// PackagingMachine object represents the packaging machine as a whole.

// right now though the packaging machine only consists of staubli robot,
// but in future projects of extending the system it is now "easy" to do so.

FUNCTION_BLOCK PackagingMachine EXTENDS UnitBaseClass
VAR_INPUT
	// initialization inputs
	inputMode		:	E_PMLProtectedUnitMode;
	inputCommand	:	E_PMLCommand;
	
	// buttons for state changes. only 6 can be used though (6 buttons in kapula)
	resetButton		AT %I*:	BIT;
	startButton		AT %I*:	BIT;
	stopButton		AT %I*:	BIT;
	holdButton		AT %I*:	BIT;
	unHoldButton	AT %I*:	BIT;
	suspendButton	AT %I*:	BIT;
	unSuspendButton	AT %I*:	BIT;
	abortButton		AT %I*:	BIT;
	clearButton		AT %I*:	BIT;
	
	// mode change buttons
	productionModeButton	AT %I*:	BIT;
	maintenanceModeButton	AT %I*:	BIT;
	manualModeButton		AT %I*:	BIT;
	
END_VAR
VAR_OUTPUT
	
END_VAR
VAR
	// container for subunits. atm only 1 subunit.
	subUnits	:	POINTER TO ARRAY[1..CONST_GV.nSubUnits] OF UnitBaseClass	:=	0;
	
	//counter for initialization
	i	:	INT;
END_VAR

IF NOT initialized THEN
	SUPER^(modeCommand:=inputMode, command:=inputCommand);
	
	IF subUnits = 0 THEN
		// subUnitsError, call setSubUnits() before PackagingMachine()
		RETURN;
	END_IF
	
	FOR i:=1 TO CONST_GV.nSubUnits BY 1 DO
		// if any of the sub units is uninitialized then the whole machine is too
		IF NOT subUnits^[i].initialized THEN
			THIS^.initialized := FALSE;
		END_IF
	END_FOR
END_IF

METHOD getSignal : INT
VAR_INPUT
END_VAR

// arranged in a way that most important ones are checked first.

// probably needs more conditions than just button signal pressed. 
// for example the statements should be ignored if machine in transition state etc.

IF abortButton THEN
	getSignal := abortSignal;
	RETURN;
	
ELSIF stopButton THEN
	getSignal := stopSignal;
	RETURN;
	
ELSIF startButton THEN
	getSignal := startSignal;
	RETURN;
	
ELSIF resetButton THEN
	getSignal := resetSignal;
	RETURN;
	
ELSIF clearButton THEN
	getSignal := clearSignal;
	RETURN;
	
ELSIF holdButton THEN
	getSignal := holdSignal;
	RETURN;
	
ELSIF unHoldButton THEN
	getSignal := unHoldSignal;
	RETURN;
	
ELSIF suspendButton THEN
	getSignal := suspendSignal;
	RETURN;
	
ELSIF unSuspendButton THEN
	getSignal := unSuspendSignal;
	RETURN;

ELSIF productionModeButton THEN
	getSignal := productionModeSignal;
	RETURN;
	
ELSIF maintenanceModeButton THEN
	getSignal := maintenanceModeSignal;
	RETURN;
	
ELSIF manualModeButton THEN
	getSignal := manualModeSignal;
	RETURN;
	
ELSE
	getSignal := -1;
	
END_IF
END_METHOD

METHOD setMode : BOOL
VAR_INPUT
	modeCommand	:	DINT;
END_VAR
VAR
	prevMode	:	E_PMLProtectedUnitMode;
END_VAR
// if any of the subUnits cannot change mode to given mode return false
FOR i:=1 TO CONST_GV.nSubUnits BY 1 DO
	IF NOT subUnits^[i].setMode(modeCommand:=modeCommand) THEN
		setMode := FALSE;
		RETURN;
	END_IF
END_FOR
SUPER^.setMode(modeCommand:=modeCommand);
setMode := TRUE;
END_METHOD


// setState method. Attempts to change the state of unit according to 
// the given input command which is a result of received user signal (startButton, stopButton ... ).

(* possible commands :	
	ePMLCommand_Undefined   := 0,
	ePMLCommand_Reset       := 1,
	ePMLCommand_Start       := 2,
	ePMLCommand_Stop        := 3,
	ePMLCommand_Hold        := 4,
	ePMLCommand_Unhold      := 5,
	ePMLCommand_Suspend     := 6,
	ePMLCommand_Unsuspend   := 7,
	ePMLCommand_Abort       := 8,
	ePMLCommand_Clear       := 9
*)

METHOD setState : BOOL
VAR_INPUT
	command	:	E_PMLCommand;
END_VAR
VAR
	prevState	:	E_PMLState;
	i			:	INT;
END_VAR
// if any of the subUnits cannot change state to given state return false
FOR i:=1 TO CONST_GV.nSubUnits BY 1 DO
	IF NOT subUnits^[i].setState(command:=command) THEN
		setState := FALSE;
		RETURN;
	END_IF
END_FOR
SUPER^.setState(command:=command);
setState := TRUE;
END_METHOD

METHOD setSubUnits : BOOL
VAR_INPUT
	inSubUnits	:	POINTER TO ARRAY[1..CONST_GV.nSubUnits] OF UnitBaseClass;
END_VAR
IF subUnits <> 0 THEN
	setSubUnits := FALSE;
	RETURN;
END_IF

subUnits := inSubUnits;
setSubUnits := TRUE;
END_METHOD

END_FUNCTION_BLOCK

(* stored: Version 1.1.0.1, ProductVersion 3.1.4022.16
   POU PackagingMachine: Id {e40f1bcf-914a-46e4-8341-5bc96b0bd344}, SpecialFunc None
   Method getSignal: Id {7e808999-f9a3-49f7-878e-9238055c1aa0}
   Method setMode: Id {6cffb050-7983-4a44-b97a-e4ac48023a93}
   Method setState: Id {c823ce98-0c6a-43f4-9247-d13fb9a55279}
   Method setSubUnits: Id {a79c9608-393b-4cda-b3b8-4d26a056df0e} *)
